FUNCTION_BLOCK FB_SomeNumber

VAR_INPUT
	
END_VAR

VAR_OUTPUT
END_VAR

VAR
	nTheNumberInQuestion : ST_DataStuff;
	
END_VAR

METHOD mRecordData : BOOL
VAR_INPUT
END_VAR
END_METHOD

METHOD mRunnerOne : BOOL

VAR_INPUT
	stInputData : ST_DataStuff;
END_VAR
// Do some calculations here, this output should differ from the other runner to track which is doing what
END_METHOD

END_FUNCTION_BLOCK

(* stored: Version 1.1.0.1, ProductVersion 3.1.4024.12
   POU FB_SomeNumber: Id {b389858d-0bd9-4a13-848a-980398a3b7c0}, SpecialFunc None
   Method mRecordData: Id {4b6172bd-1424-4ca2-95ad-7faa81a09922}
   Method mRunnerOne: Id {cce0b08b-b3a7-43d2-b62b-8c8c7f3b662a} *)
